// TIA Portal V20 export
TYPE "typeSafetyDrive"
// Safety status of drive
// stored: Access Published, IsFailsafeCompliant true, Namespace Safety
   STRUCT
      safetyFault { ExternalWritable := 'False'} : Bool;   // Safety fault in the drive 0: Fault-free operation
      stoActive { ExternalWritable := 'False'} : Bool;   // STO triggered
      ss1Active { ExternalWritable := 'False'} : Bool;   // SS1 triggered
      ss2Active { ExternalWritable := 'False'} : Bool;   // SS2 triggered
      slsActive { ExternalWritable := 'False'} : Bool;   // SLS triggered
      sosActive { ExternalWritable := 'False'} : Bool;   // SOS triggered
   END_STRUCT;
END_TYPE
